TYPE ST_Netcontactor_service :
STRUCT
	Right			: ST_service_DigitalOutInWithSafety;
	Left			: ST_service_DigitalOutInWithSafety;
END_STRUCT
END_TYPE

(* stored: Version 1.1.0.1, ProductVersion 3.1.4026.18
   DUT ST_Netcontactor_service: Id {471b76d4-04ab-4611-9854-20402008b4cd} *)
